(* CODESYS project Uppgift 11.project

Project tree, tasks and I/O mapping:
  Device : CODESYS Control Win V3, 3S - Smart Software Solutions GmbH, order no. 305021, version 3.5.10.40
    application Application
      libraries: Standard, * (System)
      task MainTask (cyclic, interval t#20ms, priority 1) calls PLC_PRG
      program PLC_PRG [ST]
      global variables GVL
      Symbols
*)

// Device/Application/GVL
{attribute 'qualified_only'}
VAR_GLOBAL
	Button: BOOL;
	SensorOpen: BOOL;
	SensorClose: BOOL;
	MotorFwd: BOOL;
	MotorRev: BOOL;
	Light: BOOL;
END_VAR

// Device/Application/PLC_PRG
PROGRAM PLC_PRG
VAR
	running: BOOL; // If the the garagerport is in the cykle or not.
	HasBeenOpend: BOOL; // if the garageport has been completly open before
	HoldDoorTImmer: TON;	// timmmer that holding the garageport open when ists completly open.
	IN_VALUE: BOOL; // the default value of garageOpenDoorTimer
	TIME_SET: TIME; // TIme thats the garageport is open
	
	LampOffTimmer: TON;
	LampOnTimmer: TON;
	TIME_SET2: TIME;
	IN_VALUE2: BOOL;
	IN_VALUE3: BOOL;
END_VAR

// Button signals
IF gvl.Button
THEN
	running := TRUE;
	HasBeenOpend := FALSE;
END_IF

// DOOR MOTOR CONTROLLER
IF running
THEN
// DOOR OPENS
	IF gvl.SensorClose
	THEN
		IF HasBeenOpend
		THEN
			running := FALSE;
		ELSE
			gvl.motorfwd := TRUE;
			gvl.MotorRev := FALSE;
	    END_IF
	END_IF
	
	// DOOR CLOSING
	IF gvl.SensorOpen
	THEN
		HasBeenOpend := TRUE;
		gvl.motorfwd := FALSE;
		
		// Timmer 
		TIME_SET := T#5S;
		IN_VALUE := TRUE;
		
		HoldDoorTImmer(IN:= IN_VALUE,PT:= TIME_SET);
		// Timmer 
		IF HoldDoorTImmer.Q
		THEN
			gvl.MotorRev := TRUE;
			IN_VALUE := FALSE;
		END_IF
	END_IF
END_IF

// Light CONTROLLER
IN_VALUE2 := TRUE;
IN_VALUE3 := TRUE;
// Time for switching lights.
TIME_SET2 := T#0.5S;

IF running
THEN
	// If sensor is open = light always on in full light
	IF gvl.SensorOpen
	THEN
		gvl.Light := TRUE;
	ELSE
		// Blingking Light
		
		LampOffTimmer(IN:= IN_VALUE2,PT:= TIME_SET2);
		IF LampOffTimmer.Q
		THEN
		// timer that set the light off if aktiv an on if not. second timmer preventing the first timer to set itself off.
			gvl.Light := FALSE;
			
			LampOnTimmer(IN:= IN_VALUE3,PT:= TIME_SET2);
			IF LampOnTimmer.Q
			THEN
				LampOnTimmer(IN:= FALSE, PT:= TIME_SET2);
				LampOffTimmer(IN:= FALSE, PT:= TIME_SET2);
			END_IF
		ELSE
			gvl.Light := TRUE;
			LampOffTimmer(IN:= TRUE,PT:= TIME_SET2);
		END_IF
	END_IF
ELSE
	gvl.Light := FALSE;
END_IF

END_PROGRAM
